{attribute 'GeneratedUsingTerminal: EL9110-0000-0016'}
{attribute addProperty BoxType "EL9110-0000-0016"}
{attribute addProperty Id "EtcSlaveTerminalBasePowerOKAT %I*PowerOK_830843C11WcStateAT %I*WcState_9091E0EB2InfoDataAT %I*InfoData_6F19DB2B2"}
{attribute addProperty CRC "3752102418"}
{attribute addProperty Size "5"}
TYPE EL9110_DFA48A12 EXTENDS EtcSlaveTerminalBase :
STRUCT
	{attribute addProperty Name "PowerOK"}
	PowerOK : PowerOK_830843C1;
	{attribute addProperty Name "WcState"}
	WcState : WcState_9091E0EB;
	{attribute addProperty Name "InfoData"}
	InfoData : InfoData_6F19DB2B;
END_STRUCT
END_TYPE

(* stored: Version 1.2.0.0, ProductVersion 3.1.4024.9
   DUT EL9110_DFA48A12: Id {5727a5d0-4b81-4cd5-b64d-557cecd33eca} *)
